// TwinCAT 3 PLC project TestPlc
// ProgramVersion: 3.1.4023.0
// libraries:
//   Tc2_Standard, * (Beckhoff Automation GmbH)
//   Tc2_System, * (Beckhoff Automation GmbH)
//   Tc3_Module, * (Beckhoff Automation GmbH)
//   tcl_AdsObjects, * (Red Rock Controls Limited)
//   tcl_UnitTestLibrary, * (Red Rock Controls Limited)
// project tree:
//   / PlcTask.TcTTO
//   POUs/ PB_TestRunner.TcPOU
//   Tasks/ PlcTask.TcTTO
// (motion and I/O tree: see PLC project tcl_adsobjects)
// real-time tasks:
//   TASK PlcTask: cycle T#10ms, priority 20, ADS port 350

CONFIGURATION TestPlc
    RESOURCE PLC ON TwinCAT3
        TASK PlcTask(INTERVAL := T#10ms, PRIORITY := 20);
        TASK PlcTask(INTERVAL := T#10ms, PRIORITY := 20);
        PROGRAM PB_TestRunner WITH PlcTask : PB_TestRunner;
        PROGRAM PB_TestRunner WITH PlcTask : PB_TestRunner;
    END_RESOURCE
END_CONFIGURATION

// ---- POUs/PB_TestRunner.TcPOU
PROGRAM PB_TestRunner
VAR
    Run : BOOL := TRUE;

    TestRunner : T_TestRunner('tcl_AdsObjects');
    
    Test_ReadBySymbolName                    : tcl_AdsObjects.Test_ReadBySymbolName(AdsPort := _AppInfo.AdsPort);
    Test_ReadWriteBySymbolName               : tcl_AdsObjects.Test_ReadWriteBySymbolName(AdsPort := _AppInfo.AdsPort);
    Test_WriteBySymbolName                   : tcl_AdsObjects.Test_WriteBySymbolName(AdsPort := _AppInfo.AdsPort);
    Test_ReadBySymbolName_KeepingHandle      : tcl_AdsObjects.Test_ReadBySymbolName_KeepingHandle(AdsPort := _AppInfo.AdsPort);
    Test_ReadWriteBySymbolName_KeepingHandle : tcl_AdsObjects.Test_ReadWriteBySymbolName_KeepingHandle(AdsPort := _AppInfo.AdsPort);
    Test_WriteBySymbolName_KeepingHandle     : tcl_AdsObjects.Test_WriteBySymbolName_KeepingHandle(AdsPort := _AppInfo.AdsPort);
END_VAR

IF Run THEN
    Run := FALSE;
    TestRunner.Initialise();
    TestRunner.AddTest(Test_ReadBySymbolName);
    TestRunner.AddTest(Test_ReadWriteBySymbolName);
    TestRunner.AddTest(Test_WriteBySymbolName);
    TestRunner.AddTest(Test_ReadBySymbolName_KeepingHandle);
    TestRunner.AddTest(Test_ReadWriteBySymbolName_KeepingHandle);
    TestRunner.AddTest(Test_WriteBySymbolName_KeepingHandle);
	TestRunner.Execute();
END_IF

TestRunner();

END_PROGRAM
